Yaskawa INFORM job: CLEAR_POS.JBI

/JOB
//NAME CLEAR_POS
///FOLDERNAME AMW2020
//POS
///NPOS 0,0,0,0,0,0
//ARGINFO
///ARGTYPE B,,,,,,,
///COMMENT
POS_SHIFT_REG







//INST
///DATE 2020/02/05 13:34
///ATTR SC,RW
///GROUP1 RB1
///LVARS 1,0,0,0,0,0,0,0
NOP
GETARG LB000 IARG#(1)
SETE P[LB000] (1) 0
SETE P[LB000] (2) 0
SETE P[LB000] (3) 0
SETE P[LB000] (4) 0
SETE P[LB000] (5) 0
SETE P[LB000] (6) 0
END
